TYPE "St_Conveyor"
VERSION : 0.1
   STRUCT
      IHM_xButtonRun : Bool;
      IHM_xStatusMotor : Int;
      iq_xError { ExternalAccessible := 'False'; ExternalVisible := 'False'; ExternalWritable := 'False'} : Bool;
      iq_iErrorType { ExternalAccessible := 'False'; ExternalVisible := 'False'; ExternalWritable := 'False'} : Int;
   END_STRUCT;

END_TYPE

